Fanuc KAREL source: ko00082.KL

PROGRAM KO00082
%STACKSIZE=65535
%PRIORITY=65535
%NOLOCKGROUP
VAR
P1 : JOINTPOS9
P2 : POSITION
F : BOOLEAN
OUT : XYZWPR
BEGIN
F=TRUE
-- UNSAFE_SOURCE_IR line 11: OUT = MIRROR(convert_jointpos9_to_xyzwprext(P1), P2, F)
END KO00082
